TYPE ST_HMI_VolumesRow  :
STRUCT
	Stage  : STRING(8);     // "T/IC", "S0", ..., "F"
    Rinse1 : REAL;
    Rinse2 : REAL;
    Wash1  : REAL;
    Wash2  : REAL;
END_STRUCT
END_TYPE

(* stored: Version 1.1.0.1, ProductVersion 3.1.4024.12
   DUT ST_HMI_VolumesRow: Id {9a0f104b-6702-4675-914e-a86335934a4b} *)
